VAR_GLOBAL
	axis1 : AXIS_REF;
END_VAR

(* stored: Version 1.1.0.1, ProductVersion 3.1.0.38
   GVL GVL: Id {783abcc7-dd7b-4a97-8da1-0353f898dda8} *)
